(* PLC project Appliances_Alarms, Actility iec61131 1.0.28, author Laurent Nicq *)
(* stored: creationDateTime 2013-06-10T10:05:45, version 1.1.0, modificationDateTime 2013-06-21T18:00:03 *)

FUNCTION_BLOCK Alarm_LimitHigh_Common
  VAR
    Dummy : BOOL;  (* to avoid Warning *)
    Alarm_High_Enable : BOOL := TRUE;
  END_VAR
  VAR_INPUT
    Alarm_High_Sensor : REAL;
    Alarm_High_Limit : REAL;
    Alarm_High_Epsilon : REAL;
  END_VAR
  VAR
    Alarm_High_Divider : REAL := 2.0;
  END_VAR
  VAR_OUTPUT
    Alarm_High_ALARM : BOOL;
  END_VAR
  VAR
    HYSTERESIS_HIGH : HYSTERESIS;
  END_VAR
  VAR  (* added by the conversion: wires and edge detectors of the diagram *)
    _DIV23_OUT : REAL;
    _SUB19_OUT : REAL;
  END_VAR

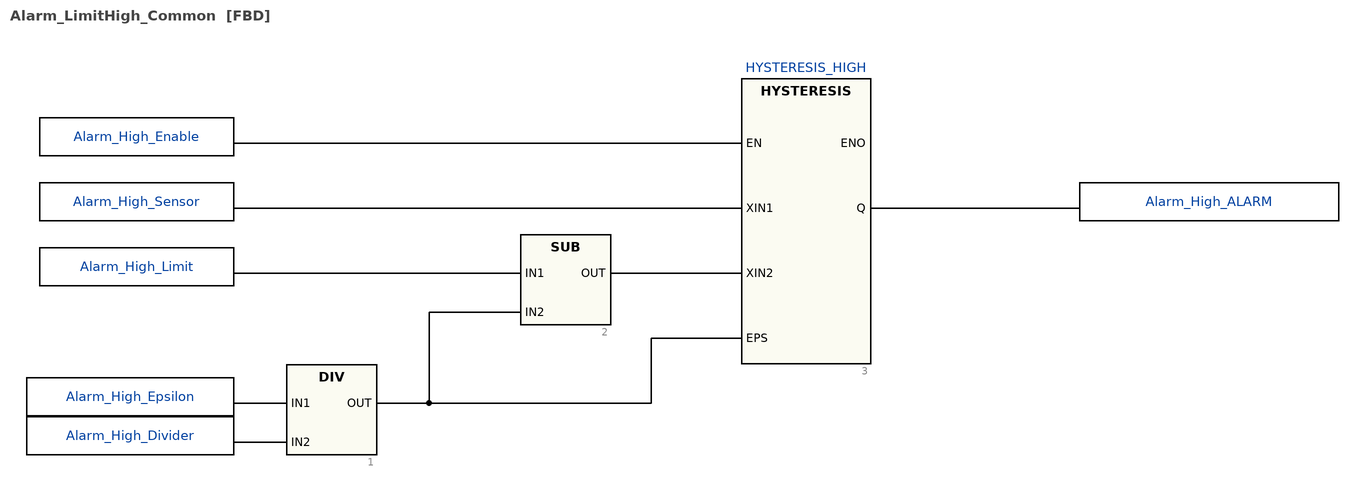
(* FBD diagram, written out as Structured Text *)
_DIV23_OUT := Alarm_High_Epsilon / Alarm_High_Divider;
_SUB19_OUT := Alarm_High_Limit - _DIV23_OUT;
HYSTERESIS_HIGH(EN := Alarm_High_Enable, XIN1 := Alarm_High_Sensor, XIN2 := _SUB19_OUT, EPS := _DIV23_OUT);
IF HYSTERESIS_HIGH.ENO THEN Alarm_High_ALARM := HYSTERESIS_HIGH.Q; END_IF;
END_FUNCTION_BLOCK

FUNCTION_BLOCK Alarm_LimitLow_Common
  VAR
    Dummy : BOOL;  (* to avoid Warning *)
    Alarm_Low_Enable : BOOL := TRUE;
  END_VAR
  VAR_INPUT
    Alarm_Low_Sensor : REAL;
    Alarm_Low_Limit : REAL;
    Alarm_Low_Epsilon : REAL;
  END_VAR
  VAR
    Alarm_Low_Divider : REAL := 2.0;
  END_VAR
  VAR_OUTPUT
    Alarm_Low_ALARM : BOOL;
  END_VAR
  VAR
    HYSTERESIS_LOW : HYSTERESIS;
  END_VAR
  VAR  (* added by the conversion: wires and edge detectors of the diagram *)
    _DIV23_OUT : REAL;
    _ADD25_OUT : REAL;
  END_VAR

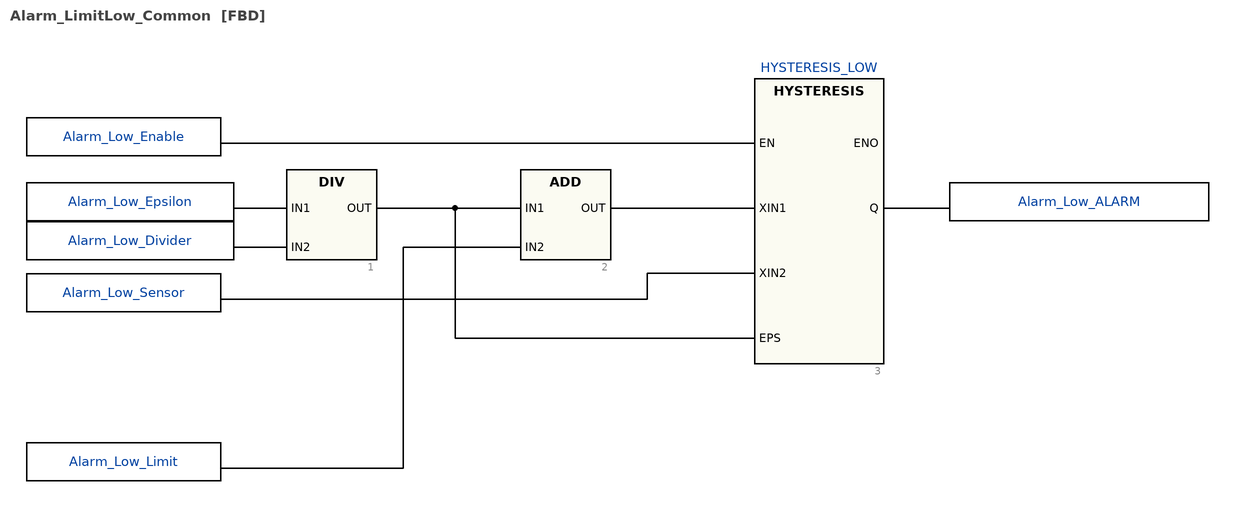
(* FBD diagram, written out as Structured Text *)
_DIV23_OUT := Alarm_Low_Epsilon / Alarm_Low_Divider;
_ADD25_OUT := _DIV23_OUT + Alarm_Low_Limit;
HYSTERESIS_LOW(EN := Alarm_Low_Enable, XIN1 := _ADD25_OUT, XIN2 := Alarm_Low_Sensor, EPS := _DIV23_OUT);
IF HYSTERESIS_LOW.ENO THEN Alarm_Low_ALARM := HYSTERESIS_LOW.Q; END_IF;
END_FUNCTION_BLOCK

FUNCTION_BLOCK Alarm_Range_Common
  VAR
    Dummy : BOOL;  (* to avoid Warning *)
    Alarm_Range_Enable : BOOL := TRUE;
  END_VAR
  VAR_INPUT
    Alarm_Range_Sensor : REAL;
    Alarm_Range_High : REAL;
    Alarm_Range_Low : REAL;
    Alarm_Range_Epsilon : REAL;
  END_VAR
  VAR
    Alarm_Range_Divider : REAL := 2.0;
  END_VAR
  VAR_OUTPUT
    Alarm_Range_ALARM : BOOL;
    Alarm_Range_ALARM_High : BOOL;
    Alarm_Range_ALARM_Low : BOOL;
  END_VAR
  VAR
    HYSTERESIS_LOW : HYSTERESIS;
    HYSTERESIS_HIGH : HYSTERESIS;
  END_VAR
  VAR  (* added by the conversion: wires and edge detectors of the diagram *)
    _DIV23_OUT : REAL;
    _SUB19_OUT : REAL;
    _ADD18_OUT : REAL;
    _OR20_OUT : BOOL;
  END_VAR

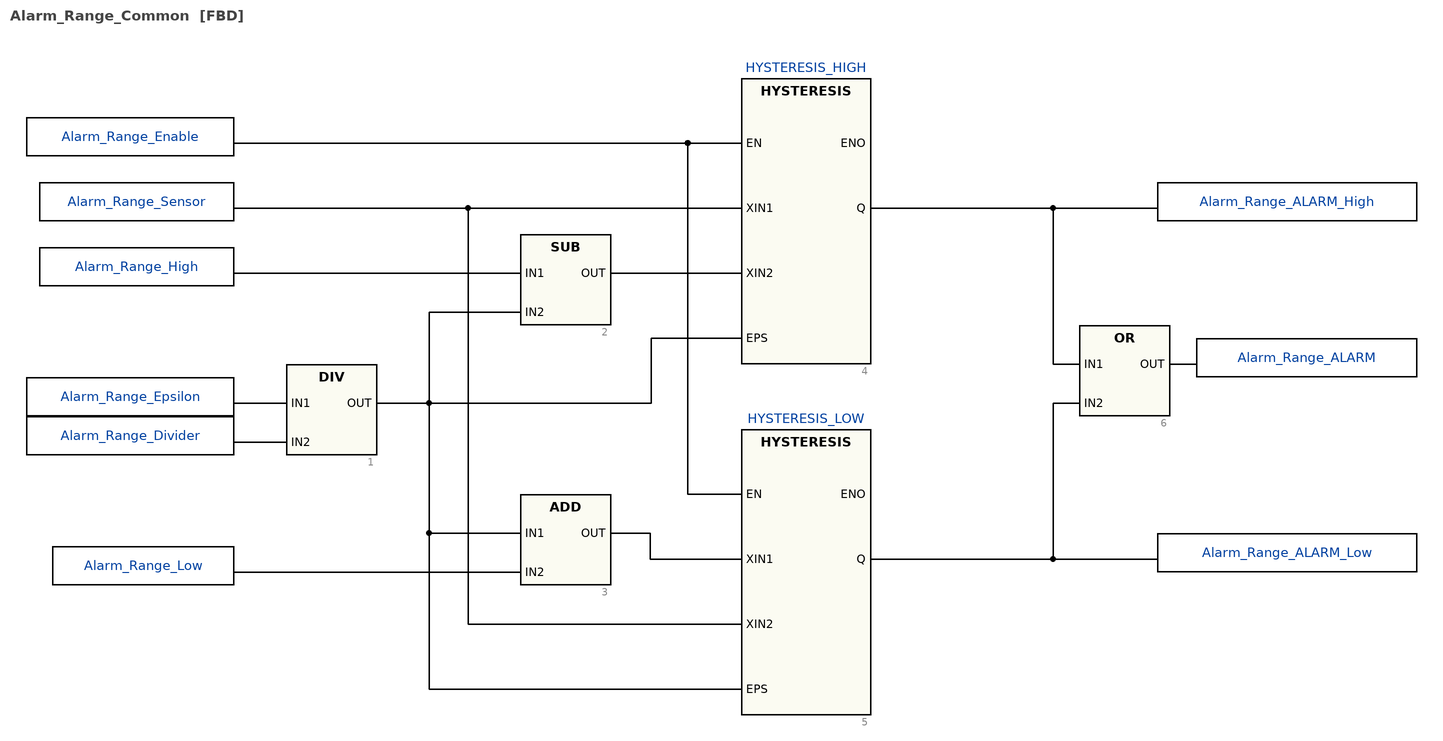
(* FBD diagram, written out as Structured Text *)
_DIV23_OUT := Alarm_Range_Epsilon / Alarm_Range_Divider;
_SUB19_OUT := Alarm_Range_High - _DIV23_OUT;
_ADD18_OUT := _DIV23_OUT + Alarm_Range_Low;
HYSTERESIS_HIGH(EN := Alarm_Range_Enable, XIN1 := Alarm_Range_Sensor, XIN2 := _SUB19_OUT, EPS := _DIV23_OUT);
HYSTERESIS_LOW(EN := Alarm_Range_Enable, XIN1 := _ADD18_OUT, XIN2 := Alarm_Range_Sensor, EPS := _DIV23_OUT);
_OR20_OUT := HYSTERESIS_HIGH.Q OR HYSTERESIS_LOW.Q;
IF HYSTERESIS_HIGH.ENO THEN Alarm_Range_ALARM_High := HYSTERESIS_HIGH.Q; END_IF;
Alarm_Range_ALARM := _OR20_OUT;
IF HYSTERESIS_LOW.ENO THEN Alarm_Range_ALARM_Low := HYSTERESIS_LOW.Q; END_IF;
END_FUNCTION_BLOCK

PROGRAM Alarm_Appliance
  VAR
    Appliance1_AlarmAny : BOOL;
    Appliance1_AlarmHigh1 : BOOL;
    Appliance1_AlarmHigh2 : BOOL;
    Appliance1_AlarmLow1 : BOOL;
    Appliance1_AlarmLow2 : BOOL;
  END_VAR
  VAR_EXTERNAL
    Appliance1_Sensor : REAL;
  END_VAR
  VAR
    Appliance1_Hyst_Epsilon : REAL := 5.0;
    Appliance1_LimitHigh : REAL := 80.0;
    Appliance1_LimitLow : REAL := 20.0;
    Alarm_Range_Limits : Alarm_Range_Common;
    Alarm_High_Limit : Alarm_LimitHigh_Common;
    Alarm_Low_Limit : Alarm_LimitLow_Common;
  END_VAR

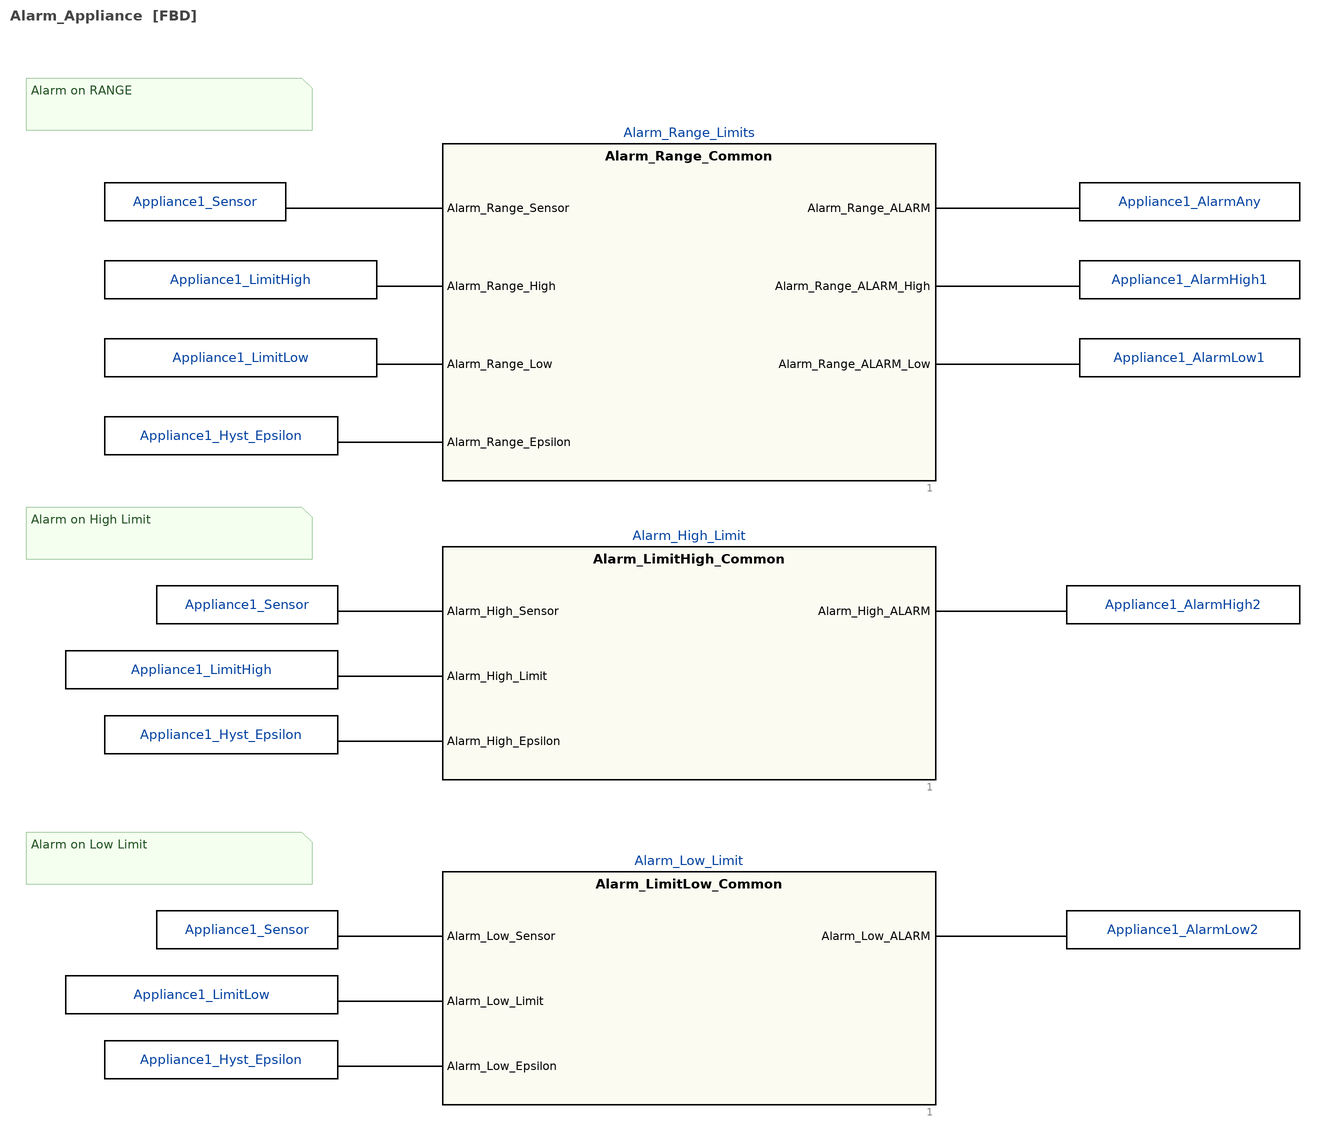
(* FBD diagram, written out as Structured Text *)
(* Alarm on RANGE *)
Alarm_Range_Limits(Alarm_Range_Sensor := Appliance1_Sensor, Alarm_Range_High := Appliance1_LimitHigh, Alarm_Range_Low := Appliance1_LimitLow, Alarm_Range_Epsilon := Appliance1_Hyst_Epsilon);
(* Alarm on High Limit *)
Alarm_High_Limit(Alarm_High_Sensor := Appliance1_Sensor, Alarm_High_Limit := Appliance1_LimitHigh, Alarm_High_Epsilon := Appliance1_Hyst_Epsilon);
(* Alarm on Low Limit *)
Alarm_Low_Limit(Alarm_Low_Sensor := Appliance1_Sensor, Alarm_Low_Limit := Appliance1_LimitLow, Alarm_Low_Epsilon := Appliance1_Hyst_Epsilon);
Appliance1_AlarmAny := Alarm_Range_Limits.Alarm_Range_ALARM;
Appliance1_AlarmHigh1 := Alarm_Range_Limits.Alarm_Range_ALARM_High;
Appliance1_AlarmLow1 := Alarm_Range_Limits.Alarm_Range_ALARM_Low;
Appliance1_AlarmHigh2 := Alarm_High_Limit.Alarm_High_ALARM;
Appliance1_AlarmLow2 := Alarm_Low_Limit.Alarm_Low_ALARM;
END_PROGRAM

FUNCTION_BLOCK Alarm_Motor_2speed_Common
  VAR
    Alarm_High_Enable : BOOL := TRUE;
  END_VAR
  VAR_INPUT
    Alarm_High_Sensor : REAL;
    Alarm_High_Limit1 : REAL;
    Alarm_High_Limit2 : REAL;
    Alarm_High_Epsilon : REAL;
  END_VAR
  VAR
    Alarm_High_Divider : REAL := 2.0;
  END_VAR
  VAR_OUTPUT
    Alarm_High_ALARM : BOOL;  (* Any Threshold reached *)
    Alarm_High_SPEED : BOOL;  (* False: Level1 True: Level2 *)
  END_VAR
  VAR
    HYSTERESIS_HIGH : HYSTERESIS;
    HYSTERESIS0 : HYSTERESIS;
  END_VAR
  VAR  (* added by the conversion: wires and edge detectors of the diagram *)
    _DIV23_OUT : REAL;
    _SUB19_OUT : REAL;
    _SUB6_OUT : REAL;
    _NOT28_OUT : BOOL;
    _OR25_OUT : BOOL;
  END_VAR

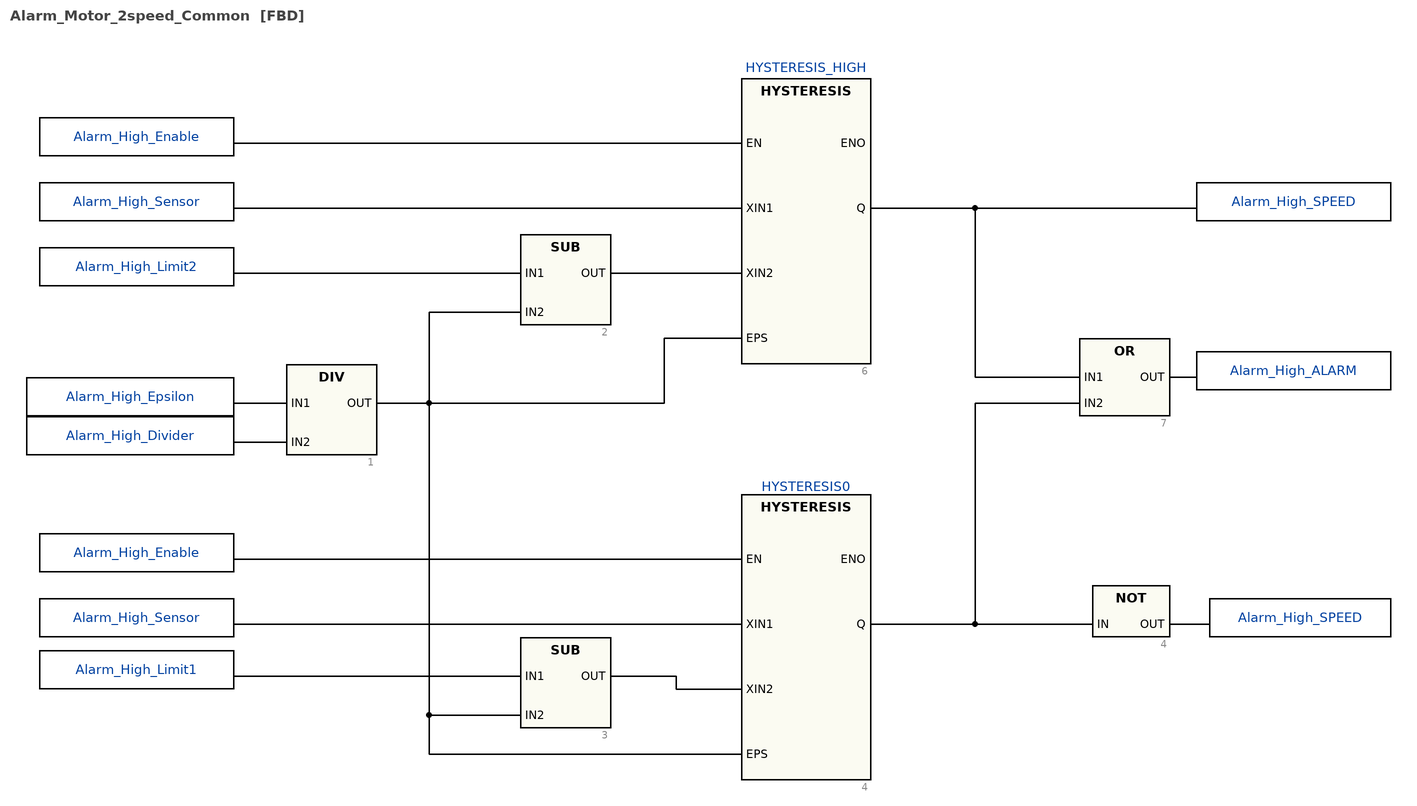
(* FBD diagram, written out as Structured Text *)
_DIV23_OUT := Alarm_High_Epsilon / Alarm_High_Divider;
_SUB19_OUT := Alarm_High_Limit2 - _DIV23_OUT;
_SUB6_OUT := Alarm_High_Limit1 - _DIV23_OUT;
HYSTERESIS0(EN := Alarm_High_Enable, XIN1 := Alarm_High_Sensor, XIN2 := _SUB6_OUT, EPS := _DIV23_OUT);
_NOT28_OUT := NOT HYSTERESIS0.Q;
HYSTERESIS_HIGH(EN := Alarm_High_Enable, XIN1 := Alarm_High_Sensor, XIN2 := _SUB19_OUT, EPS := _DIV23_OUT);
_OR25_OUT := HYSTERESIS_HIGH.Q OR HYSTERESIS0.Q;
IF HYSTERESIS_HIGH.ENO THEN Alarm_High_SPEED := HYSTERESIS_HIGH.Q; END_IF;
Alarm_High_ALARM := _OR25_OUT;
Alarm_High_SPEED := _NOT28_OUT;
END_FUNCTION_BLOCK

PROGRAM Ventilation
  VAR
    Start_Ventilation : BOOL := TRUE;
    Ventilation_Information : STRING := '';
    Ventilation_Mode : DINT := -1;  (* 0: Stop 1: Forced 2: Automatic *)
    Ventilation_Type : BOOL := TRUE;  (* False: single speed True: two speed *)
    Ventilate_ON : BOOL;
    Ventilate_Speed : BOOL;  (* False = Speed1 True=Speed2 *)
  END_VAR
  VAR_EXTERNAL
    Humidity_Sensor : REAL;  (* Simulated *)
  END_VAR
  VAR
    Humidity_Threshold1 : REAL := 60.0;  (* Limit Speed1 *)
    Humidity_Threshold2 : REAL := 80.0;  (* Limit Speed2 *)
    Humidity_Hyst_Eps : REAL := 5.0;  (* Hysteresis band *)
    Speed1_Humidity : Alarm_LimitHigh_Common;
    Speed2_Humidity : Alarm_Motor_2speed_Common;
  END_VAR

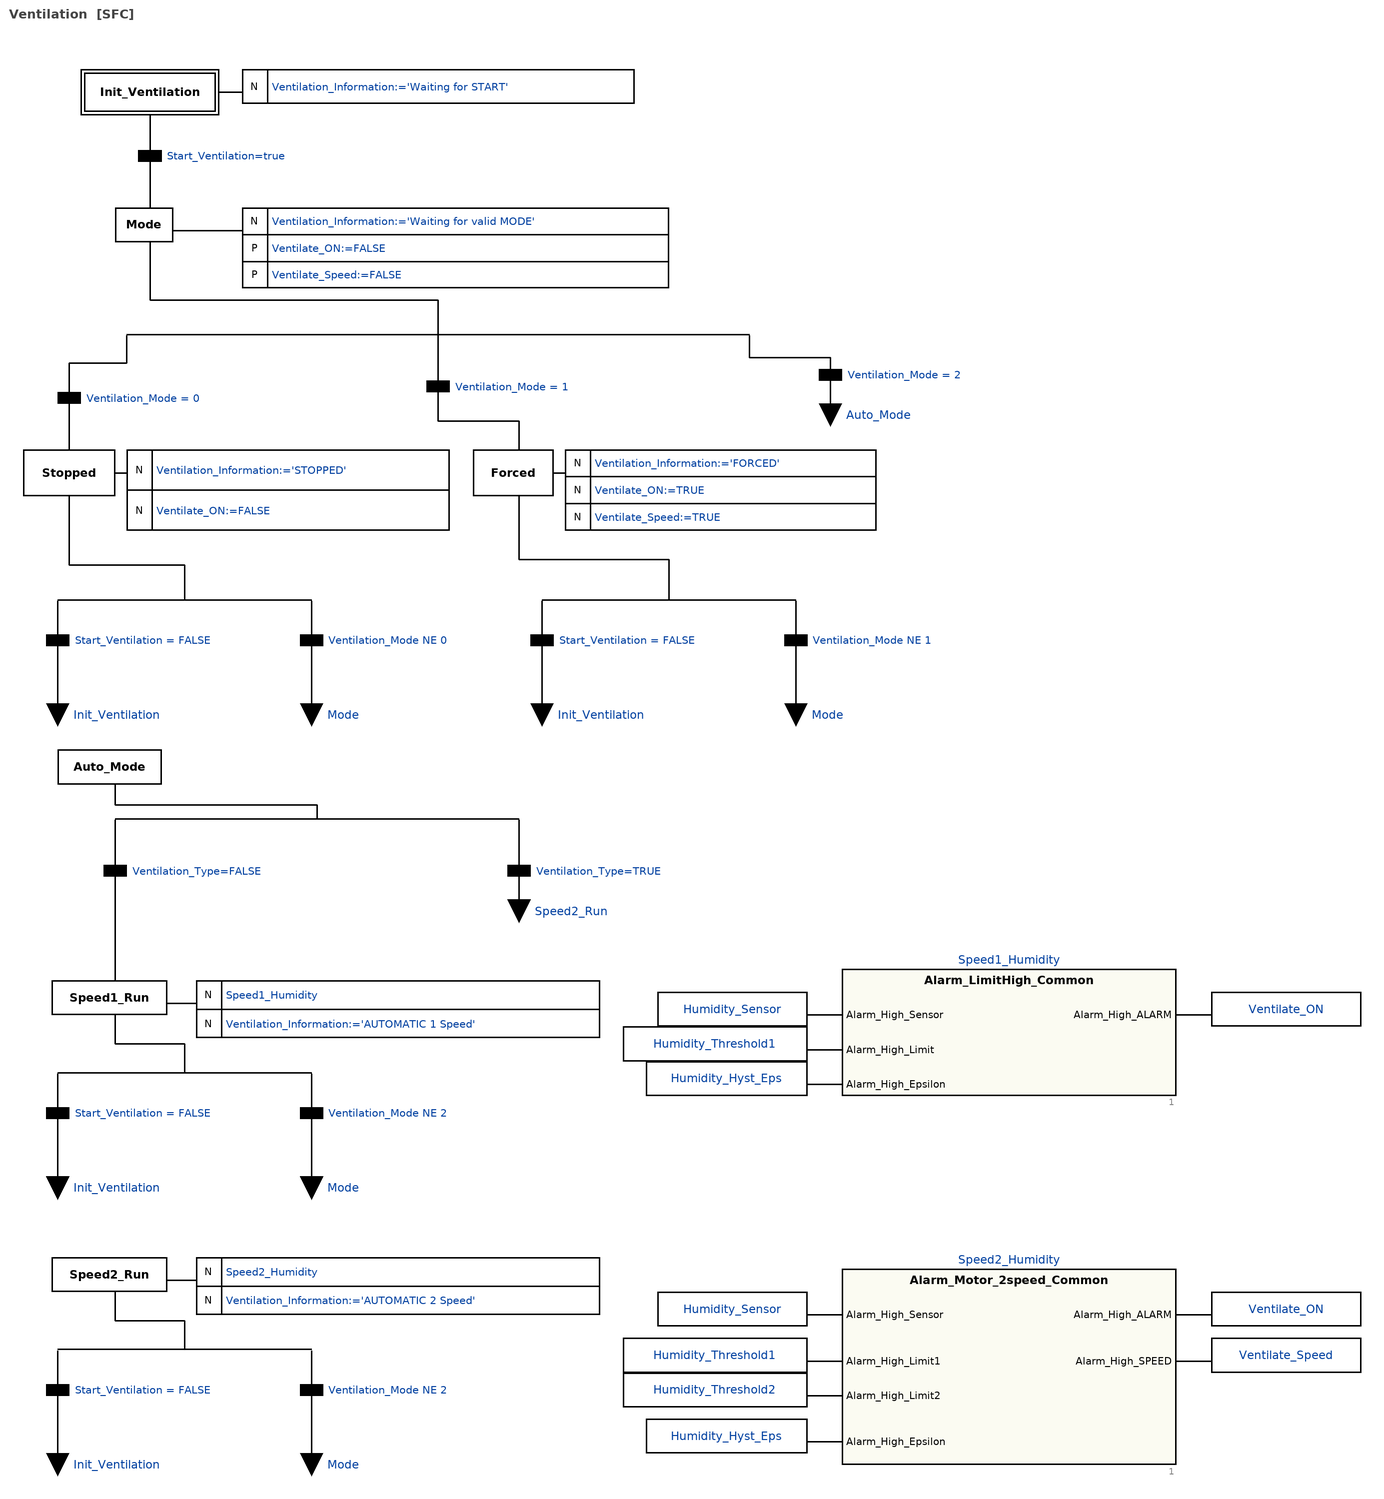
INITIAL_STEP Init_Ventilation:
  INIT_VENTILATION_INLINE1(N);
  COMPUTE_FUNCTION_BLOCKS(S);
END_STEP
ACTION INIT_VENTILATION_INLINE1:
  Ventilation_Information:='Waiting for START'
END_ACTION
TRANSITION FROM Init_Ventilation TO Mode
  := Start_Ventilation=true;
END_TRANSITION
STEP Mode:
  MODE_INLINE2(N);
  MODE_INLINE3(P);
  MODE_INLINE4(P);
END_STEP
ACTION MODE_INLINE2:
  Ventilation_Information:='Waiting for valid MODE'
END_ACTION
ACTION MODE_INLINE3:
  Ventilate_ON:=FALSE
END_ACTION
ACTION MODE_INLINE4:
  Ventilate_Speed:=FALSE
END_ACTION
TRANSITION FROM Mode TO Stopped
  := Ventilation_Mode = 0;
END_TRANSITION
TRANSITION FROM Mode TO Forced
  := Ventilation_Mode = 1;
END_TRANSITION
TRANSITION FROM Mode TO Auto_Mode
  := Ventilation_Mode = 2;
END_TRANSITION
STEP Stopped:
  STOPPED_INLINE5(N);
  STOPPED_INLINE6(N);
END_STEP
ACTION STOPPED_INLINE5:
  Ventilation_Information:='STOPPED'
END_ACTION
ACTION STOPPED_INLINE6:
  Ventilate_ON:=FALSE
END_ACTION
TRANSITION FROM Stopped TO Init_Ventilation
  := Start_Ventilation = FALSE;
END_TRANSITION
TRANSITION FROM Stopped TO Mode
  := Ventilation_Mode NE 0;
END_TRANSITION
STEP Forced:
  FORCED_INLINE7(N);
  FORCED_INLINE8(N);
  FORCED_INLINE9(N);
END_STEP
ACTION FORCED_INLINE7:
  Ventilation_Information:='FORCED'
END_ACTION
ACTION FORCED_INLINE8:
  Ventilate_ON:=TRUE
END_ACTION
ACTION FORCED_INLINE9:
  Ventilate_Speed:=TRUE
END_ACTION
TRANSITION FROM Forced TO Init_Ventilation
  := Start_Ventilation = FALSE;
END_TRANSITION
TRANSITION FROM Forced TO Mode
  := Ventilation_Mode NE 1;
END_TRANSITION
STEP Auto_Mode:
END_STEP
TRANSITION FROM Auto_Mode TO Speed1_Run
  := Ventilation_Type=FALSE;
END_TRANSITION
TRANSITION FROM Auto_Mode TO Speed2_Run
  := Ventilation_Type=TRUE;
END_TRANSITION
STEP Speed1_Run:
  Speed1_Humidity(N);
  SPEED1_RUN_INLINE10(N);
END_STEP
ACTION SPEED1_RUN_INLINE10:
  Ventilation_Information:='AUTOMATIC 1 Speed'
END_ACTION
TRANSITION FROM Speed1_Run TO Init_Ventilation
  := Start_Ventilation = FALSE;
END_TRANSITION
TRANSITION FROM Speed1_Run TO Mode
  := Ventilation_Mode NE 2;
END_TRANSITION
STEP Speed2_Run:
  Speed2_Humidity(N);
  SPEED2_RUN_INLINE11(N);
END_STEP
ACTION SPEED2_RUN_INLINE11:
  Ventilation_Information:='AUTOMATIC 2 Speed'
END_ACTION
TRANSITION FROM Speed2_Run TO Init_Ventilation
  := Start_Ventilation = FALSE;
END_TRANSITION
TRANSITION FROM Speed2_Run TO Mode
  := Ventilation_Mode NE 2;
END_TRANSITION
ACTION COMPUTE_FUNCTION_BLOCKS:  (* blocks drawn on the SFC sheet *)
  Speed1_Humidity(Alarm_High_Sensor := Humidity_Sensor, Alarm_High_Limit := Humidity_Threshold1, Alarm_High_Epsilon := Humidity_Hyst_Eps);
  Speed2_Humidity(Alarm_High_Sensor := Humidity_Sensor, Alarm_High_Limit1 := Humidity_Threshold1, Alarm_High_Limit2 := Humidity_Threshold2, Alarm_High_Epsilon := Humidity_Hyst_Eps);
  Ventilate_ON := Speed1_Humidity.Alarm_High_ALARM;
  Ventilate_ON := Speed2_Humidity.Alarm_High_ALARM;
  Ventilate_Speed := Speed2_Humidity.Alarm_High_SPEED;
END_ACTION
END_PROGRAM

PROGRAM Simulation
  VAR
    Start_Simul : BOOL := true;
    WAVE_Gen : WAVE_GENERATOR;
    Signal_Type : INT := 1;  (* Generate Sinus *)
    Signal_Amplitude : REAL := 100.0;  (* from 0 to 100 *)
    Signal_Average : REAL := 50.0;  (* from 0 to 100 *)
    Signal_Period : REAL := 30;
  END_VAR
  VAR_EXTERNAL
    Appliance1_Sensor : REAL;
    Humidity_Sensor : REAL;
  END_VAR

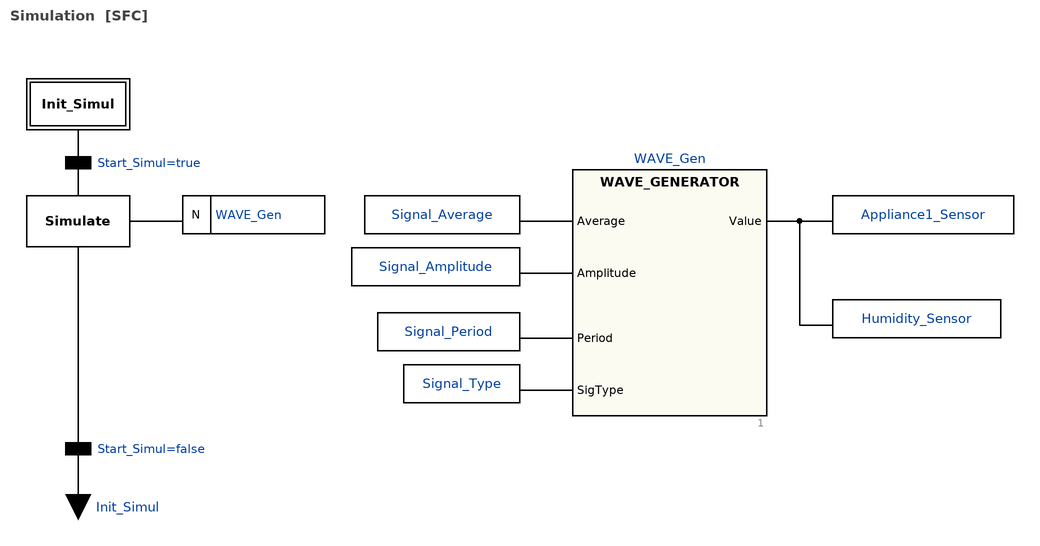
INITIAL_STEP Init_Simul:
  COMPUTE_FUNCTION_BLOCKS(S);
END_STEP
TRANSITION FROM Init_Simul TO Simulate
  := Start_Simul=true;
END_TRANSITION
STEP Simulate:
  WAVE_Gen(N);
END_STEP
TRANSITION FROM Simulate TO Init_Simul
  := Start_Simul=false;
END_TRANSITION
ACTION COMPUTE_FUNCTION_BLOCKS:  (* blocks drawn on the SFC sheet *)
  WAVE_Gen(Average := Signal_Average, Amplitude := Signal_Amplitude, Period := Signal_Period, SigType := Signal_Type);
  Appliance1_Sensor := WAVE_Gen.Value;
  Humidity_Sensor := WAVE_Gen.Value;
END_ACTION
END_PROGRAM

CONFIGURATION config
  RESOURCE resource_main ON PLC
    VAR_GLOBAL
      Appliance1_Sensor : REAL := 50.0;
      Humidity_Sensor : REAL := 50.0;
    END_VAR
    TASK Sampling_Slow(INTERVAL := T#1s0ms, PRIORITY := 0);
    TASK Sampling_Fast(INTERVAL := T#500ms, PRIORITY := 0);
    PROGRAM Simulator WITH Sampling_Slow : Simulation;
    PROGRAM Appliance WITH Sampling_Fast : Alarm_Appliance;
    PROGRAM Ventil WITH Sampling_Fast : Ventilation;
  END_RESOURCE
END_CONFIGURATION
